% RSLogix 500 project Logic_Functions.RSS, saved by version 8.30.01.01 %
PROJECT "UNTITLED"    % processor: Bul.1763 MicroLogix 1100 Series A %

PROGRAM FILES
  LAD 2   5 rungs

DATA FILES
  O0 OUTPUT  4 elements
  I1 INPUT  6 elements
  S2 STATUS  66 elements
  B3 BINARY  1 elements
  T4 TIMER  1 elements
  C5 COUNTER  1 elements
  R6 CONTROL  1 elements
  N7 INTEGER  1 elements
  F8 FLOAT  1 elements

LADDER 2
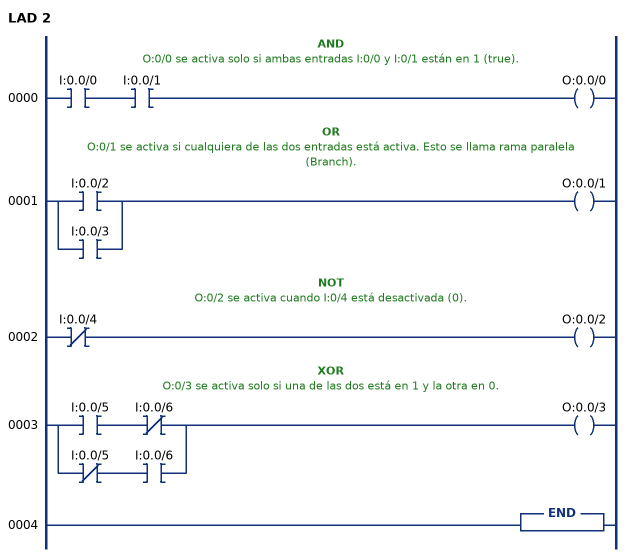
% Rung: 0 %
% TITLE: AND %
% O:0/0 se activa solo si ambas entradas I:0/0 y I:0/1 están en 1 (true). %
SOR XIC I:0.0/0 XIC I:0.0/1 OTE O:0.0/0 EOR
% Rung: 1 %
% TITLE: OR %
% O:0/1 se activa si cualquiera de las dos entradas está activa. Esto se llama rama paralela (Branch). %
SOR BST XIC I:0.0/2 NXB XIC I:0.0/3 BND OTE O:0.0/1 EOR
% Rung: 2 %
% TITLE: NOT %
% O:0/2 se activa cuando I:0/4 está desactivada (0). %
SOR XIO I:0.0/4 OTE O:0.0/2 EOR
% Rung: 3 %
% TITLE: XOR %
% O:0/3 se activa solo si una de las dos está en 1 y la otra en 0. %
SOR BST XIC I:0.0/5 XIO I:0.0/6 NXB XIO I:0.0/5 XIC I:0.0/6 BND OTE O:0.0/3 EOR
% Rung: 4 %
SOR END EOR
